% RSLogix 500 project PRACTISE-7.RSS, saved by version 8.30.00.16 %
PROJECT "UNTITLED"    % processor: Bul.1763 MicroLogix 1100 Series A %

PROGRAM FILES
  LAD 2   10 rungs

DATA FILES
  O0 OUTPUT  4 elements
  I1 INPUT  6 elements
  S2 STATUS  66 elements
  B3 BINARY  1 elements
  T4 TIMER  1 elements
  C5 COUNTER  1 elements
  R6 CONTROL  1 elements
  N7 INTEGER  30 elements
  F8 FLOAT  1 elements

LADDER 2
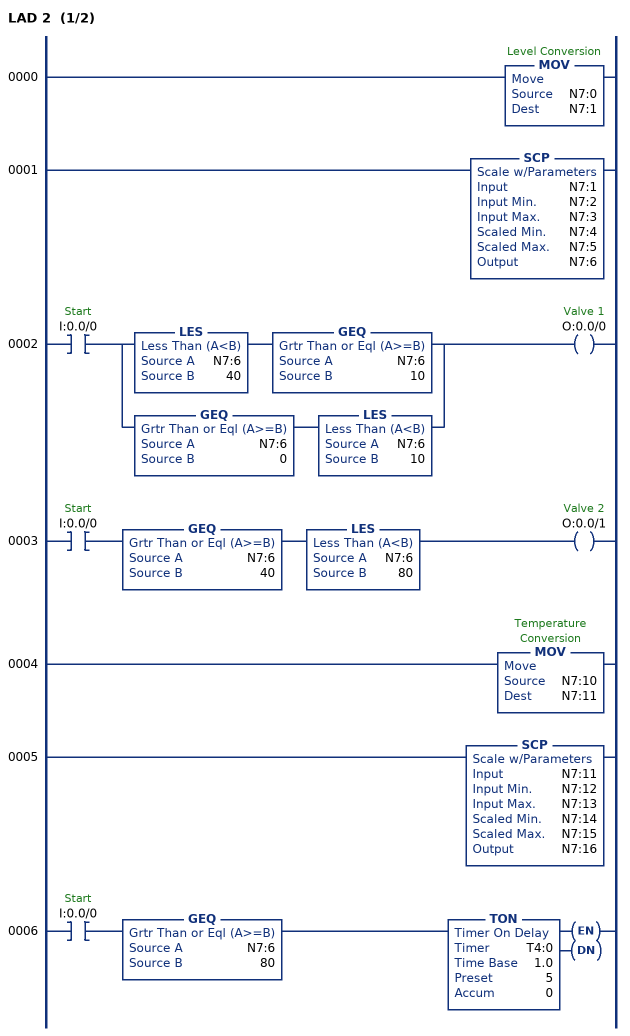
% Rung: 0 %
SOR MOV N7:0 N7:1 EOR
%   N7:1  "Level Conversion" %
% Rung: 1 %
SOR SCP N7:1 N7:2 N7:3 N7:4 N7:5 N7:6 EOR
%   N7:1  "Level Conversion" %
% Rung: 2 %
SOR XIC I:0.0/0 BST LES N7:6 40 GEQ N7:6 10 NXB GEQ N7:6 0 LES N7:6 10 BND OTE O:0.0/0 EOR
%   I:0.0/0  "Start" %
%   O:0.0/0  "Valve 1" %
% Rung: 3 %  % edit flag set %
SOR XIC I:0.0/0 GEQ N7:6 40 LES N7:6 80 OTE O:0.0/1 EOR
%   I:0.0/0  "Start" %
%   O:0.0/1  "Valve 2" %
% Rung: 4 %
SOR MOV N7:10 N7:11 EOR
%   N7:10  MOV %
%   N7:11  "Temperature Conversion" %
% Rung: 5 %
SOR SCP N7:11 N7:12 N7:13 N7:14 N7:15 N7:16 EOR
%   N7:11  "Temperature Conversion" %
% Rung: 6 %  % edit flag set %
SOR XIC I:0.0/0 GEQ N7:6 80 TON T4:0 1.0 5 0 EOR
%   I:0.0/0  "Start" %

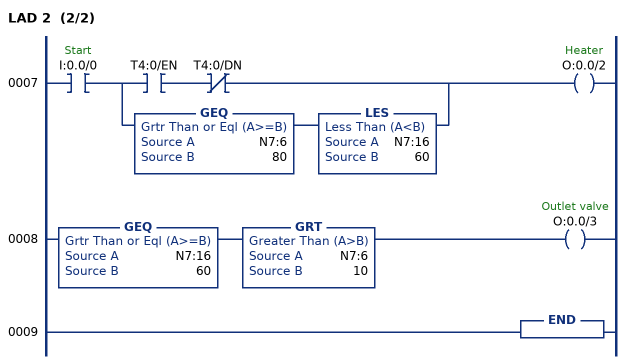
% Rung: 7 %
SOR XIC I:0.0/0 BST XIC T4:0/EN XIO T4:0/DN NXB GEQ N7:6 80 LES N7:16 60 BND OTE O:0.0/2 EOR
%   I:0.0/0  "Start" %
%   O:0.0/2  "Heater" %
% Rung: 8 %
SOR GEQ N7:16 60 GRT N7:6 10 OTE O:0.0/3 EOR
%   O:0.0/3  "Outlet valve" %
% Rung: 9 %
SOR END EOR

OTHER DOCUMENTED ADDRESSES
  CPY  
  I:0.0/1  "Analog Level Sensor"

DATA TABLE (non-zero values as saved)
DATA T4
% .PRE .ACC %
% T4:0 % 5 0
DATA N7
% N7:0 % 1000 0 20000 0 100 0 0 0 0 0
% N7:10 % 1000 0 0 2000 0 100 0 0 0 0
